(* CODESYS project TANQUE.project

Project tree, tasks and I/O mapping:
  Device : CODESYS Control Win V3, 3S - Smart Software Solutions GmbH, order no. 305021, version 3.5.11.30
    application Application
      libraries: Standard, * (System)
      task MainTask (cyclic, interval t#20ms, priority 1) calls PLC_PRG
      program PLC_PRG [ST]
*)

// Device/Application/PLC_PRG
PROGRAM PLC_PRG
VAR
   START : BOOL;       // inicia o processo
   STOP  : BOOL;       // para tudo
   LT1   : BOOL;       // sensor de nivel 1
   LT2   : BOOL;       // sensor de nivel 2
   LT3   : BOOL;       // sensor de nivel 3
   MV1   : BOOL;
   MV2   : BOOL;
   EST   : BOOL;      // esteira
   STIR  : BOOL;      // motor stir
   P1    : BOOL;      // passo 1
   P2    : BOOL;      // passo 2
   P3    : BOOL;      // passo 3
   P4    : BOOL;      // passo 4
   P5    : BOOL;      // passo 5
   P6    : BOOL;      // passo 6
   CV1   : WORD;
   PULSO : BOOL;
   PULSO1 : BOOL;
   CT1Q   : BOOL;
   ET1    : TIME;
   ET2    : TIME;
   CT1    : CTU;
   TP1   : TP;
   TP2   : TP;
   ET3   : TIME;
   RT1 :  R_TRIG;
   RT2 : R_TRIG;
   RT3 : R_TRIG;
   FT1 : F_TRIG;
   FT2 : F_TRIG;
   TON1 : TON;
   TON2 : TON;
   ET4 : TIME;
   END_VAR

P1 := (START OR P1) AND NOT(STOP);
P2 := (NOT(LT1) OR P2) AND P1 AND NOT(P6);
P3 := (LT2 OR P3) AND P2;
P4 := (LT3 OR P4) AND P3;
RT1(CLK := P6);
RT2(CLK := STIR);
CT1(CU := P4 AND RT2.Q, RESET := RT1.Q, PV := 3, CV => CV1);
P5 := P4 AND CT1Q;
P6 := P5 AND NOT(LT1);
MV1 := P2 AND NOT(P3);
MV2 := P5 AND NOT(P6);  
EST := P3 AND NOT(P4);
STIR := P4 AND NOT(P5) AND PULSO;
FT1(CLK := TP2.Q);
RT3(CLK := P4);
TP1(IN := TP2.Q OR P4,PT := T#10S,Q => PULSO,ET => ET1);
FT2(CLK := TP1.Q);
TP2(IN := TP1.Q ,PT := T#55S,Q => PULSO,ET => ET2);
TON1(IN := P4 AND NOT(TON2.Q),PT := T#5S,Q => PULSO1,ET => ET3);
TON2(IN := TON1.Q,PT := T#10S,ET => ET4);

END_PROGRAM
